SUBAPPLICATION rastend (* Subapplication Type *)
  (* Standard: 61499-2 *)
  (* Version 1.0, 2024-10-23, franz *)
  PACKAGE FBs::Uebungen::Uebung_103::subapp;
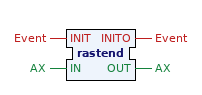
  EVENT_INPUT
    INIT; (* Initialization Request *)
  END_EVENT
  EVENT_OUTPUT
    INITO; (* Initialization Confirm *)
  END_EVENT
  SOCKETS
    IN : AX;
  END_SOCKETS
  PLUGS
    OUT : AX;
  END_PLUGS
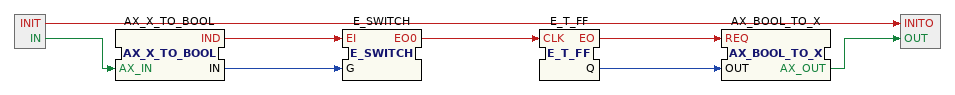
  (* soll beim Loslassen gestarte t werden ! *)
  FBS
    E_T_FF : E_T_FF;
    E_SWITCH : E_SWITCH;
    AX_X_TO_BOOL : AX_X_TO_BOOL;
    AX_BOOL_TO_X : AX_BOOL_TO_X;
  END_FBS
  EVENT_CONNECTIONS
    INIT TO INITO;
    E_SWITCH.EO0 TO E_T_FF.CLK;
    E_T_FF.EO TO AX_BOOL_TO_X.REQ;
    AX_X_TO_BOOL.IND TO E_SWITCH.EI;
  END_CONNECTIONS
  DATA_CONNECTIONS
    E_T_FF.Q TO AX_BOOL_TO_X.OUT;
    AX_X_TO_BOOL.IN TO E_SWITCH.G;
  END_CONNECTIONS
  ADAPTER_CONNECTIONS
    IN TO AX_X_TO_BOOL.AX_IN;
    AX_BOOL_TO_X.AX_OUT TO OUT;
  END_CONNECTIONS
END_SUBAPPLICATION
